// Mitsubishi GX Works2 project: 240409_지연간격동작회로   PLC: Q03UDV

PROGRAM MAIN
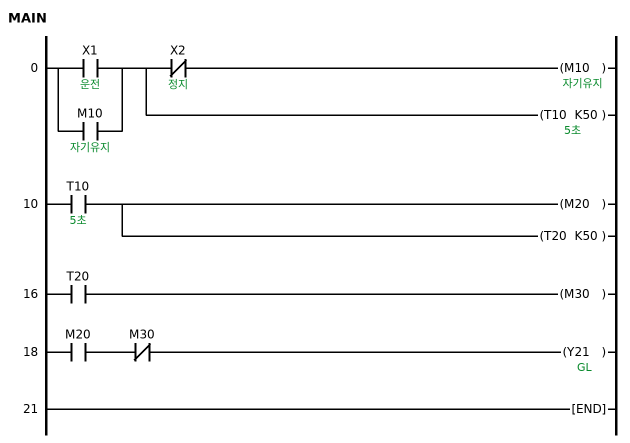
0     LD      X1  ; 운전
      OR      M10  ; 자기유지
      MPS
      ANI     X2  ; 정지
      OUT     M10  ; 자기유지
      MPP
      OUT     T10 K50  ; 5초
10    LD      T10  ; 5초
      OUT     M20
      OUT     T20 K50
16    LD      T20
      OUT     M30
18    LD      M20
      ANI     M30
      OUT     Y21  ; GL
21    END
END_PROGRAM

// device comments not shown above
X0  ; 정지
Y22  ; 정지
